Yaskawa INFORM job: RRR.JBI

/JOB
//NAME RRR
//POS
///NPOS 0,0,0,0,0,0
//INST
///DATE 2024/01/09 19:56
///ATTR SC,RW,RJ
////FRAME ROBOT
///GROUP1 RB1,BS1
NOP
END
